KUKA KRL program: chk_w5_grp2_clo.src

&ACCESS RVO1
&COMMENT Actros Z2.1_Z2.2
DEF chk_w5_grp2_clo( )
; Check gripper ACTROS CLOSE Z2.1 Z2.2
;//---- Start User-------


$TIMER[10] = 0
$TIMER_STOP[10] = FALSE

WAIT FOR ($IN[8] AND $IN[10])
WAIT FOR (NOT $IN[7] AND NOT $IN[9])

$TIMER_STOP[10] = TRUE
$TIMER[10] = 0

;//---- End User---------
END
